PROGRAM PRG_Test
VAR
	FC_AddTests : FC_Add_Test;
END_VAR

TCUnit.RUN();

END_PROGRAM

(* stored: Version 1.1.0.1
   POU PRG_Test: Id {d6b2cab2-1c70-4756-9b9a-734830e723c7}, SpecialFunc None *)
